// TIA Portal V17 export
// export: Created 2025-06-26T06:33:55.8470365Z, ExportSetting WithDefaults, DisplayName Totally Integrated Automation Portal, DisplayVersion V17 Update 8, DisplayName TIA Portal Openness, DisplayVersion V17 Update 8, DisplayName TIA Portal Version Control Interface, DisplayVersion V17, DisplayName STEP 7 Professional, DisplayVersion V17 Update 8, DisplayName STEP 7 Safety, DisplayVersion V17 Update 6, DisplayName WinCC Advanced, DisplayVersion V17 Update 8
FUNCTION_BLOCK "ModbusRTUMaster"   // FB7, FBD
TITLE = Modbus RTU Master
{ S7_Optimized_Access := 'TRUE' }
VERSION : 0.1
// Sequence communication to several nodes. Each node is just added as more states to the state machine. There are better ways to do this but this will do for now.
// stored: AutoNumber true, IsIECCheckEnabled false, IsRetainMemResEnabled false, MemoryReserve 0, SetENOAutomatically false, UDAEnableTagReadback false
   VAR_INPUT
      bFirstCycle : Bool;
      bStart : Bool;
   END_VAR
   VAR_OUTPUT
      Done { ExternalAccessible := 'False'; ExternalVisible := 'False'; ExternalWritable := 'False'} : Bool;
      Initialised : Bool;   // 1 = successful init
   END_VAR
   VAR
      InitReq : Bool;
      InitErrorCode : Word;
      InitSuccess : Bool;
      ReadReq : Bool;
      MasterDoneStored : Bool;
      MasterStatus_stored : Word;
      MasterDone : Bool;
      MasterError : Bool;
      MasterBusy : Bool;
      MasterStatus : Word;
      State : USInt;
      Wait : TON_TIME;
      Node1CommCycles { S7_SetPoint := 'True'} : UDInt;
      Node2CommCycles : UDInt;
      Node10CommCycles : UDInt;
      Node20CommCycles : UDInt;
   END_VAR
   VAR_TEMP
      InitDone : Bool;
      InitError : Bool;
      InitStatus : Word;
   END_VAR
BEGIN

REGION Network 1 (SCL): Init modbus
   // NOTE: The DB at Modbus_Master's DATA_PTR pin must have "Optimized Access" disabled in its properties.
   // Modbus_Master's MODE input: (S7-1200 Programmable controller system manual, P. 1199 (A5E02486680-AM)
   // MODE 0 : Read Modbus address 1 to 9999, 10001 to 19999 as bits, 30001 to 39999, 40001 to 49999 as words
   // MODE 104 : Read Modbus address 0 to 65535 as words
   // Mode 1 : Write Modbus address 1 to 9999 as bits, 40001 to 49999 as words, 2 or more at a time
   // Mode 2 : As above but 1 or more at a time

   CASE #State OF
       0:  // IDLE
           IF #bStart = TRUE THEN
               #Done := FALSE;
               #InitReq := TRUE;
               #State := 1;
               #Node1CommCycles := 0;
               #Node2CommCycles := 0;
               #Node20CommCycles := 0;
           END_IF;
       1:  // INIT (runs once, not once every comm cycle)

           // For some reason, the duplex mode has to be set manually, and before the init block runs. 
           // Source: Siemens demo project for CM1241. Doesn't work without.
           "Modbus_Comm_Load_DB".MODE := 4;
           // REQ can only be high for one cycle. Wait 100ms (RESP_TO ) for slave response
           "Modbus_Comm_Load_DB"(REQ := #InitReq, 
                                 PORT := "Local~Modbus_RTU", 
                                 BAUD := 19200, 
                                 PARITY := 0, 
                                 FLOW_CTRL := 0, 
                                 RTS_ON_DLY := 0, 
                                 RTS_OFF_DLY := 0, 
                                 RESP_TO := 100, 
                                 MB_DB := "Modbus_Master_DB".MB_DB,
                                 DONE => #InitDone,
                                 ERROR => #InitError,
                                 STATUS => #InitStatus);
           #InitReq := FALSE;
           IF #InitDone THEN
               #InitSuccess := TRUE;
               #InitErrorCode := 0;
               #State := 4;
           ELSIF #InitError THEN
               #InitSuccess := FALSE;
               #InitErrorCode := #InitStatus;
               #State := 1;
           END_IF;
           #Initialised := #InitSuccess;
   (* ### Rewrite this for the actual nodes in the communication
       3: // Done
           // Optional wait between cycles
           //#Wait(IN := TRUE, PT := T#1ms);
           //IF #Wait.Q = TRUE THEN
           //    #Done := TRUE;
           //    #State := 4;
           //END_IF;
           #Done := TRUE;
           #State := 4;

       4: // Read Node 1
           "Modbus_Master_DB"(REQ := TRUE,
                               MB_ADDR := 1, 
                               MODE := 0, 
                               DATA_ADDR := 40009, 
                               DATA_LEN := 4,
                               DATA_PTR := P#DB10.DBX0.0 WORD 8,
                               DONE => #MasterDone,
                               BUSY => #MasterBusy,
                               ERROR => #MasterError,
                               STATUS => #MasterStatus);
           IF #MasterError = TRUE THEN 
               #MasterStatus_stored := #MasterStatus;
               "TA_State".%X0 := FALSE;
               #State := 6;
           ELSIF #MasterDone = TRUE THEN
               #MasterStatus := 0;
               "TA_State".%X0 := TRUE;
               "TA1_Rx".SW := "MasterData".dataPtr.data[0];
               "TA1_Rx".Act1 := "MasterData".dataPtr.data[1];
               "TA1_Rx".Act2 := "MasterData".dataPtr.data[2];
               "TA1_Rx".DataIO_12 := "MasterData".dataPtr.data[3];
               #State := 5;
           END_IF;
       5: // Write Node 1
           "MasterData".dataPtr.data[0] := "TA1_Tx".CW;
           "MasterData".dataPtr.data[1] := "TA1_Tx".Ref1;
           "MasterData".dataPtr.data[2] := "TA1_Tx".Ref2;
           "Modbus_Master_DB"(REQ := TRUE,
                               MB_ADDR := 1, 
                               MODE := 1, 
                               DATA_ADDR := 40001, 
                               DATA_LEN := 3,
                               DATA_PTR := P#DB10.DBX0.0 WORD 8,
                               DONE => #MasterDone,
                               BUSY => #MasterBusy,
                               ERROR => #MasterError,
                               STATUS => #MasterStatus);
           IF #MasterError = TRUE THEN 
               #MasterStatus_stored := #MasterStatus;
               "TA_State".%X0 := FALSE;
               #State := 6;
           ELSIF #MasterDone = TRUE THEN
               #MasterStatus := 0;
               "TA_State".%X0 := TRUE;
               #State := 6;
               #Node1CommCycles := #Node1CommCycles + 1;
           END_IF;
       6: // Read Node 2
           "Modbus_Master_DB"(REQ := TRUE,
                               MB_ADDR := 2, 
                               MODE := 0, 
                               DATA_ADDR := 40009, 
                               DATA_LEN := 4,
                               DATA_PTR := P#DB10.DBX0.0 WORD 8,
                               DONE => #MasterDone,
                               BUSY => #MasterBusy,
                               ERROR => #MasterError,
                               STATUS => #MasterStatus);
           IF #MasterError = TRUE THEN 
               #MasterStatus_stored := #MasterStatus;
               "TA_State".%X1 := FALSE;
               #State := 8;
           ELSIF #MasterDone = TRUE THEN
               #MasterStatus := 0;
               "TA_State".%X1 := TRUE;
               "TA2_Rx".SW :="MasterData".dataPtr.data[0];
               "TA2_Rx".Act1 := "MasterData".dataPtr.data[1];
               "TA2_Rx".Act2 := "MasterData".dataPtr.data[2];
               "TA2_Rx".DataIO_12 := "MasterData".dataPtr.data[3];
               #State := 7;
           END_IF;
       7: // Write Node 2
           "MasterData".dataPtr.data[0] := "TA2_Tx".CW;
           "MasterData".dataPtr.data[1] := "TA2_Tx".Ref1;
           "MasterData".dataPtr.data[2] := "TA2_Tx".Ref2;
           "Modbus_Master_DB"(REQ := TRUE,
                               MB_ADDR := 2, 
                               MODE := 1, 
                               DATA_ADDR := 40001, 
                               DATA_LEN := 3,
                               DATA_PTR := P#DB10.DBX0.0 WORD 8,
                               DONE => #MasterDone,
                               BUSY => #MasterBusy,
                               ERROR => #MasterError,
                               STATUS => #MasterStatus);
           IF #MasterError = TRUE THEN 
               #MasterStatus_stored := #MasterStatus;
               "TA_State".%X1 := FALSE;
               #State := 8;
           ELSIF #MasterDone = TRUE THEN
               #MasterStatus := 0;
               "TA_State".%X1 := TRUE;
               #State := 8;
               #Node2CommCycles := #Node2CommCycles + 1;   
           END_IF;

       8: // Read Node 10
           "Modbus_Master_DB"(REQ := TRUE,
                               MB_ADDR := 10, 
                               MODE := 0, 
                               DATA_ADDR := 40009, 
                               DATA_LEN := 4,
                               DATA_PTR := P#DB10.DBX0.0 WORD 8,
                               DONE => #MasterDone,
                               BUSY => #MasterBusy,
                               ERROR => #MasterError,
                               STATUS => #MasterStatus);
           IF #MasterError = TRUE THEN 
               #MasterStatus_stored := #MasterStatus;
               "TA_State".%X2 := FALSE;
               #State := 10;
           ELSIF #MasterDone = TRUE THEN
               #MasterStatus := 0;
               "TA_State".%X2 := TRUE;
               "TA10_Rx".SW :="MasterData".dataPtr.data[0];
               "TA10_Rx".Act1 := "MasterData".dataPtr.data[1];
               "TA10_Rx".Act2 := "MasterData".dataPtr.data[2];
               "TA10_Rx".DataIO_12 := "MasterData".dataPtr.data[3];
               #State := 9;
           END_IF;
       9: // Write Node 10
           "MasterData".dataPtr.data[0] := "TA10_Tx".CW;
           "MasterData".dataPtr.data[1] := "TA10_Tx".Ref1;
           "MasterData".dataPtr.data[2] := "TA10_Tx".Ref2;
           "Modbus_Master_DB"(REQ := TRUE,
                               MB_ADDR := 10, 
                               MODE := 1, 
                               DATA_ADDR := 40001, 
                               DATA_LEN := 3,
                               DATA_PTR := P#DB10.DBX0.0 WORD 8,
                               DONE => #MasterDone,
                               BUSY => #MasterBusy,
                               ERROR => #MasterError,
                               STATUS => #MasterStatus);
           IF #MasterError = TRUE THEN 
               #MasterStatus_stored := #MasterStatus;
               "TA_State".%X2 := FALSE;
               #State := 10;
           ELSIF #MasterDone = TRUE THEN
               "TA_State".%X2 := TRUE;
               #MasterStatus := 0;
               #State := 10;
               #Node10CommCycles := #Node10CommCycles + 1;   
           END_IF;

       10: // Read Node 20
           "Modbus_Master_DB"(REQ := TRUE,
                               MB_ADDR := 20, 
                               MODE := 104, 
                               DATA_ADDR := 16#0, 
                               DATA_LEN := 2,
                               DATA_PTR := P#DB10.DBX0.0 WORD 8,
                               DONE => #MasterDone,
                               BUSY => #MasterBusy,
                               ERROR => #MasterError,
                               STATUS => #MasterStatus);
           IF #MasterError = TRUE THEN 
               #MasterStatus_stored := #MasterStatus;
               "TA_State".%X7 := FALSE;
               #State := 3;
           ELSIF #MasterDone = TRUE THEN
               "TA_State".%X7 := TRUE;
               #MasterStatus := 0;
               "CVM1" := "MasterData".dataPtr.data[0];
               "CVM2" := "MasterData".dataPtr.data[1];
               #Node20CommCycles := #Node20CommCycles + 1;
               #State := 3;
           END_IF;

       // More nodes can go here, remember to jump to State 3 last.
   *)
   END_CASE;
END_REGION
END_FUNCTION_BLOCK
